FUNCTION_BLOCK FB_Cinta_SFC // EXTENDS FB_Module_SFC
VAR_INPUT
	ctInp: S_ControllerInput;
	//TK_1: TIME;					// Temporizador empujador tapa
	//k1: BOOL; 					// Sensor de empujador tapa delante
END_VAR
VAR_OUTPUT
	ctOut: S_ControllerOutput;
	//K_1: BOOL; (* Actuador de empujador tapa avanza *)
	//FM : BOOL; 
END_VAR

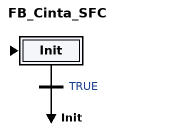
INITIAL_STEP Init:
END_STEP
TRANSITION FROM Init TO Init
    := TRUE;
END_TRANSITION

END_FUNCTION_BLOCK

(* stored: Version 1.1.0.1, ProductVersion 3.1.4024.11
   POU FB_Cinta_SFC: Id {7a4e0e2e-bc1d-4eb2-80cf-952f4dd5e6da}, SpecialFunc None *)
